// TIA Portal project "washing machine-1s" (V16)

(* hardware
DEVICE "S7-1200 station_1"  S7-1200 Station
   slot 0: "Rack_0"  S7-1200 Rack  Rack  V1.0
   slot 1: "PLC_1"  CPU 1212C AC/DC/Rly  6ES7 212-1BE40-0XB0  V4.0
*)

// ===== PLC "PLC_1"  CPU 1212C AC/DC/Rly =====

VAR_GLOBAL   // PLC tag table "Default tag table"
   "operate" AT %I0.1 : Bool;
   "KF" AT %Q0.0 : Bool;
   "KR" AT %Q0.1 : Bool;
   "Tag_1" AT %M0.0 : Bool;
   "Tag_2" AT %M0.5 : Bool;
   "Tag_3" AT %M0.6 : Bool;
END_VAR

// folder: System blocks/Program resources

DATA_BLOCK "C1"   // DB1
{ S7_Optimized_Access := 'TRUE' }
AUTHOR : Simatic
FAMILY : IEC
NAME : CNTR
VERSION : 1.0
// stored: InstanceOfName IEC_COUNTER
"IEC_COUNTER"
BEGIN
END_DATA_BLOCK

// folder: (top level)

ORGANIZATION_BLOCK "Main"   // OB1, LAD, ProgramCycle
TITLE = "Main Program Sweep (Cycle)"
{ S7_Optimized_Access := 'TRUE' }
VERSION : 0.1
   VAR_INPUT
      Initial_Call : Bool;   // Initial call of this OB
      Remanence : Bool;   // =True, if remanent data are available
   END_VAR
   VAR_TEMP   // added for the SCL form of the ladder/FBD networks
      _w1 : Bool;
   END_VAR
BEGIN

REGION Network 1
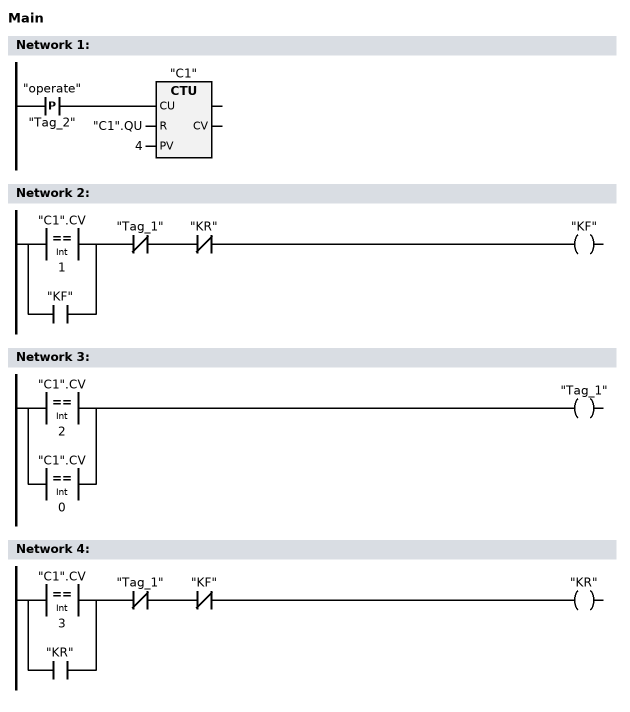
   #_w1 := "operate" AND NOT "Tag_2";   // rising edge of "operate"
   "Tag_2" := "operate";
   "C1".CTU(CU := #_w1, R := "C1".QU, PV := 4);
END_REGION

REGION Network 2
   RUNG wire#powerrail
      { S7_Templates := "SrcType := Int" } EQ_Contact(in1 := "C1".CV, in2 := 1)
      wire#w1
      I_Contact( "Tag_1" )
      I_Contact( "KR" )
      Coil( "KF" )
   END_RUNG
   RUNG wire#powerrail
      Contact( "KF" )
   END_RUNG wire#w1
   // the same network as SCL:
   "KF" := (("C1".CV = 1) OR "KF") AND NOT "Tag_1" AND NOT "KR";
END_REGION

REGION Network 3
   RUNG wire#powerrail
      { S7_Templates := "SrcType := Int" } EQ_Contact(in1 := "C1".CV, in2 := 2)
      wire#w1
      Coil( "Tag_1" )
   END_RUNG
   RUNG wire#powerrail
      { S7_Templates := "SrcType := Int" } EQ_Contact(in1 := "C1".CV, in2 := 0)
   END_RUNG wire#w1
   // the same network as SCL:
   "Tag_1" := ("C1".CV = 2) OR ("C1".CV = 0);
END_REGION

REGION Network 4
   RUNG wire#powerrail
      { S7_Templates := "SrcType := Int" } EQ_Contact(in1 := "C1".CV, in2 := 3)
      wire#w1
      I_Contact( "Tag_1" )
      I_Contact( "KF" )
      Coil( "KR" )
   END_RUNG
   RUNG wire#powerrail
      Contact( "KR" )
   END_RUNG wire#w1
   // the same network as SCL:
   "KR" := (("C1".CV = 3) OR "KR") AND NOT "Tag_1" AND NOT "KF";
END_REGION
END_ORGANIZATION_BLOCK